Fanuc TP program (LS listing): B003.LS

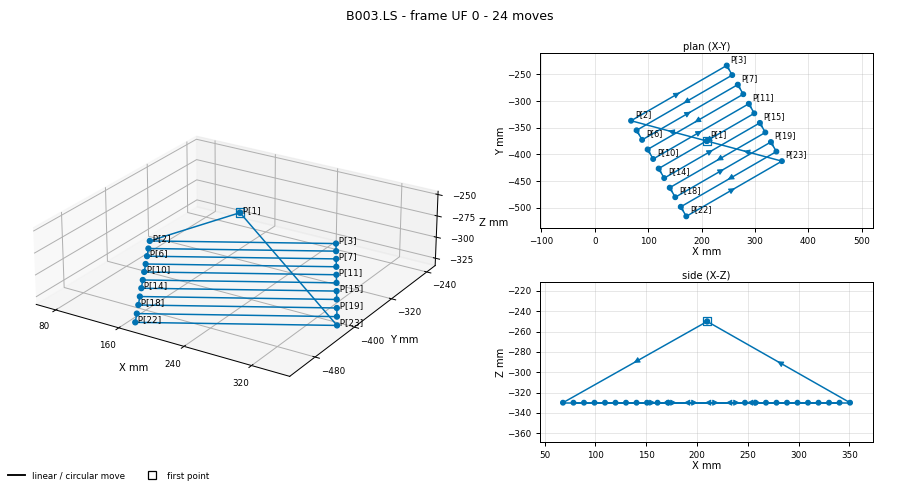
[picture p0: tool path of B003.LS in frame UF 0, 24 of 24 moves have a stored position in this frame; points joined in program order, loops and branches not executed]
/PROG  B003.LS
/ATTR
OWNER       = MNEDITOR;
COMMENT     = "";
PROG_SIZE   = 636;
CREATE      = DATE 23-01-07  TIME 11:59:14;
MODIFIED    = DATE 23-01-07  TIME 12:02:18;
FILE_NAME   = ;
VERSION     = 0;
LINE_COUNT  = 4;
MEMORY_SIZE = 992;
PROTECT     = READ_WRITE;
TCD:  STACK_SIZE	= 0,
      TASK_PRIORITY	= 50,
      TIME_SLICE	= 0,
      BUSY_LAMP_OFF	= 0,
      ABORT_REQUEST	= 0,
      PAUSE_REQUEST	= 0;
DEFAULT_GROUP	= 1,*,*,*,*;
CONTROL_CODE	= 00000000 00000000;
/MN
   1:J P[1] 100% FINE    ;
   2:L P[2] 100mm/sec CNT100    ;
   3:L P[3] 100mm/sec CNT100    ;
   4:L P[4] 100mm/sec CNT100    ;
   5:L P[5] 100mm/sec CNT100    ;
   6:L P[6] 100mm/sec CNT100    ;
   7:L P[7] 100mm/sec CNT100    ;
   8:L P[8] 100mm/sec CNT100    ;
   9:L P[9] 100mm/sec CNT100    ;
   10:L P[10] 100mm/sec CNT100    ;
   11:L P[11] 100mm/sec CNT100    ;
   12:L P[12] 100mm/sec CNT100    ;
   13:L P[13] 100mm/sec CNT100    ;
   14:L P[14] 100mm/sec CNT100    ;
   15:L P[15] 100mm/sec CNT100    ;
   16:L P[16] 100mm/sec CNT100    ;
   17:L P[17] 100mm/sec CNT100    ;
   18:L P[18] 100mm/sec CNT100    ;
   19:L P[19] 100mm/sec CNT100    ;
   20:L P[20] 100mm/sec CNT100    ;
   21:L P[21] 100mm/sec CNT100    ;
   22:L P[22] 100mm/sec CNT100    ;
   23:L P[23] 100mm/sec CNT100    ;
   24:L P[24] 100mm/sec CNT100    ;
/POS
P[1]{
   GP1:
	UF : 0, UT : 6,		CONFIG : 'N U T, 0, 0, 0',
	X =  210.000  mm,	Y =   -375.000  mm,	Z =   -250.000  mm,
	W =  90.000 deg,	P =   0.000 deg,	R =   90.000 deg
};
P[2]{
   GP1:
	UF : 0, UT : 6,		CONFIG : 'N U T, 0, 0, 0',
	X =  68.008  mm,	Y =   -336.981  mm,	Z =   -330.000  mm,
	W =  90.000 deg,	P =   0.000 deg,	R =   90.000 deg
};
P[3]{
   GP1:
	UF : 0, UT : 6,		CONFIG : 'N U T, 0, 0, 0',
	X =  247.225  mm,	Y =   -233.502  mm,	Z =   -330.000  mm,
	W =  90.000 deg,	P =   0.000 deg,	R =   90.000 deg
};
P[4]{
   GP1:
	UF : 0, UT : 6,		CONFIG : 'N U T, 0, 0, 0',
	X =  257.571  mm,	Y =   -251.421  mm,	Z =   -330.000  mm,
	W =  90.000 deg,	P =   0.000 deg,	R =   90.000 deg
};
P[5]{
   GP1:
	UF : 0, UT : 6,		CONFIG : 'N U T, 0, 0, 0',
	X =  78.354  mm,	Y =   -354.900  mm,	Z =   -330.000  mm,
	W =  90.000 deg,	P =   0.000 deg,	R =   90.000 deg
};
P[6]{
   GP1:
	UF : 0, UT : 6,		CONFIG : 'N U T, 0, 0, 0',
	X =  88.700  mm,	Y =   -372.819  mm,	Z =   -330.000  mm,
	W =  90.000 deg,	P =   0.000 deg,	R =   90.000 deg
};
P[7]{
   GP1:
	UF : 0, UT : 6,		CONFIG : 'N U T, 0, 0, 0',
	X =  267.918  mm,	Y =   -269.340  mm,	Z =   -330.000  mm,
	W =  90.000 deg,	P =   0.000 deg,	R =   90.000 deg
};
P[8]{
   GP1:
	UF : 0, UT : 6,		CONFIG : 'N U T, 0, 0, 0',
	X =  278.264  mm,	Y =   -287.259  mm,	Z =   -330.000  mm,
	W =  90.000 deg,	P =   0.000 deg,	R =   90.000 deg
};
P[9]{
   GP1:
	UF : 0, UT : 6,		CONFIG : 'N U T, 0, 0, 0',
	X =  99.047  mm,	Y =   -390.738  mm,	Z =   -330.000  mm,
	W =  90.000 deg,	P =   0.000 deg,	R =   90.000 deg
};
P[10]{
   GP1:
	UF : 0, UT : 6,		CONFIG : 'N U T, 0, 0, 0',
	X =  109.393  mm,	Y =   -408.657  mm,	Z =   -330.000  mm,
	W =  90.000 deg,	P =   0.000 deg,	R =   90.000 deg
};
P[11]{
   GP1:
	UF : 0, UT : 6,		CONFIG : 'N U T, 0, 0, 0',
	X =  288.610  mm,	Y =   -305.178  mm,	Z =   -330.000  mm,
	W =  90.000 deg,	P =   0.000 deg,	R =   90.000 deg
};
P[12]{
   GP1:
	UF : 0, UT : 6,		CONFIG : 'N U T, 0, 0, 0',
	X =  298.957  mm,	Y =   -323.097  mm,	Z =   -330.000  mm,
	W =  90.000 deg,	P =   0.000 deg,	R =   90.000 deg
};
P[13]{
   GP1:
	UF : 0, UT : 6,		CONFIG : 'N U T, 0, 0, 0',
	X =  119.739  mm,	Y =   -426.576  mm,	Z =   -330.000  mm,
	W =  90.000 deg,	P =   0.000 deg,	R =   90.000 deg
};
P[14]{
   GP1:
	UF : 0, UT : 6,		CONFIG : 'N U T, 0, 0, 0',
	X =  130.086  mm,	Y =   -444.495  mm,	Z =   -330.000  mm,
	W =  90.000 deg,	P =   0.000 deg,	R =   90.000 deg
};
P[15]{
   GP1:
	UF : 0, UT : 6,		CONFIG : 'N U T, 0, 0, 0',
	X =  309.303  mm,	Y =   -341.016  mm,	Z =   -330.000  mm,
	W =  90.000 deg,	P =   0.000 deg,	R =   90.000 deg
};
P[16]{
   GP1:
	UF : 0, UT : 6,		CONFIG : 'N U T, 0, 0, 0',
	X =  319.649  mm,	Y =   -358.935  mm,	Z =   -330.000  mm,
	W =  90.000 deg,	P =   0.000 deg,	R =   90.000 deg
};
P[17]{
   GP1:
	UF : 0, UT : 6,		CONFIG : 'N U T, 0, 0, 0',
	X =  140.432  mm,	Y =   -462.414  mm,	Z =   -330.000  mm,
	W =  90.000 deg,	P =   0.000 deg,	R =   90.000 deg
};
P[18]{
   GP1:
	UF : 0, UT : 6,		CONFIG : 'N U T, 0, 0, 0',
	X =  150.778  mm,	Y =   -480.333  mm,	Z =   -330.000  mm,
	W =  90.000 deg,	P =   0.000 deg,	R =   90.000 deg
};
P[19]{
   GP1:
	UF : 0, UT : 6,		CONFIG : 'N U T, 0, 0, 0',
	X =  329.996  mm,	Y =   -376.855  mm,	Z =   -330.000  mm,
	W =  90.000 deg,	P =   0.000 deg,	R =   90.000 deg
};
P[20]{
   GP1:
	UF : 0, UT : 6,		CONFIG : 'N U T, 0, 0, 0',
	X =  340.342  mm,	Y =   -394.774  mm,	Z =   -330.000  mm,
	W =  90.000 deg,	P =   0.000 deg,	R =   90.000 deg
};
P[21]{
   GP1:
	UF : 0, UT : 6,		CONFIG : 'N U T, 0, 0, 0',
	X =  161.125  mm,	Y =   -498.252  mm,	Z =   -330.000  mm,
	W =  90.000 deg,	P =   0.000 deg,	R =   90.000 deg
};
P[22]{
   GP1:
	UF : 0, UT : 6,		CONFIG : 'N U T, 0, 0, 0',
	X =  171.471  mm,	Y =   -516.171  mm,	Z =   -330.000  mm,
	W =  90.000 deg,	P =   0.000 deg,	R =   90.000 deg
};
P[23]{
   GP1:
	UF : 0, UT : 6,		CONFIG : 'N U T, 0, 0, 0',
	X =  350.688  mm,	Y =   -412.693  mm,	Z =   -330.000  mm,
	W =  90.000 deg,	P =   0.000 deg,	R =   90.000 deg
};
P[24]{
   GP1:
	UF : 0, UT : 6,		CONFIG : 'N U T, 0, 0, 0',
	X =  210.000  mm,	Y =   -375.000  mm,	Z =   -250.000  mm,
	W =  90.000 deg,	P =   0.000 deg,	R =   90.000 deg
};
/END
